// TIA Portal V16 export
// export: Created 2021-07-12T14:47:16.6551787Z, ExportSetting WithDefaults, DisplayName Totally Integrated Automation Portal, DisplayVersion V16, DisplayName TIA Portal Version Control Interface, DisplayVersion V16, DisplayName TIA Portal Openness, DisplayVersion V16, DisplayName STEP 7 Professional, DisplayVersion V16, DisplayName STEP 7 Safety, DisplayVersion V16, DisplayName WinCC Professional, DisplayVersion V16
DATA_BLOCK "LSimaHydTO_MC_ForceControl_DB"   // DB1
AUTHOR : APC_ERLF
FAMILY : LSimaHydTO
VERSION : 1.0
// stored: AutoNumber true, DBAccessibleFromOPCUA true, InstanceOfName LSimaHydTO_MC_ForceControl, InstanceOfType FB
"LSimaHydTO_MC_ForceControl"
   // VAR_INPUT
   //    execute : Bool;
   //    forceControlProfile : UInt;
   //    mode : DInt;
   //    forceProfileMode : DInt;
   //    conditionMode : DInt;
   //    compareMode : DInt;
   //    conditionValue : LReal;
   //    forceValue : LReal;
   //    forceDerivedValue : LReal;
   //    velocityLimitingValue : LReal;
   // END_VAR
   // VAR_OUTPUT
   //    done { ExternalWritable := 'False'} : Bool;
   //    inForceControl { ExternalWritable := 'False'} : Bool;
   //    busy { ExternalWritable := 'False'} : Bool;
   //    commandAborted { ExternalWritable := 'False'} : Bool;
   //    error { ExternalWritable := 'False'} : Bool;
   //    errorID { ExternalWritable := 'False'} : Word;
   // END_VAR
   // VAR_IN_OUT
   //    axis : "LSimaHydTO_typeAxisData";
   // END_VAR
   // VAR
   //    statFBState { ExternalAccessible := 'False'; ExternalVisible := 'False'; ExternalWritable := 'False'} : DInt;
   //    statCommandID { ExternalAccessible := 'False'; ExternalVisible := 'False'; ExternalWritable := 'False'} : UDInt;
   //    statCmdState { ExternalAccessible := 'False'; ExternalVisible := 'False'; ExternalWritable := 'False'} : Word;
   //    statExecuteOld { ExternalAccessible := 'False'; ExternalVisible := 'False'; ExternalWritable := 'False'} : Bool;
   // END_VAR
BEGIN
END_DATA_BLOCK
